// TIA Portal V20 export
TYPE "LER_typeStatusGeneral"
// stored: Access Published
   STRUCT
      stageWidth : LReal := 244.14;
      stageWidthOffset : LReal := 33.18;
      stageGap : LReal := 1.0;
      stageHeight : LReal := 350.0;
      lineSpeed : LReal;
      startSpeedCpm : LReal := 5.0;
      accTime : LReal := 2.0;
      dccTime : LReal := 2.0;
      countOffset : LReal;
      nowValue : LReal;
      nowCount : DInt;
      stopValue : LReal;
      stopCount : DInt;
      stopTarget : LReal;
      repeatMode : Bool;
      onlyStackMode : Bool;
      anodeToDo : Bool;
      cathodeToDo : Bool;
   END_STRUCT;
END_TYPE
